# EPICS autosave request: apps/xpsMotorApp/Db/hpsSvtTopScan.req
$(PREF)hps:svt_top:motor:scan1.P1PA
$(PREF)hps:svt_top:motor:scan1.P1SM
$(PREF)hps:svt_top:motor:scan1.P1SP
$(PREF)hps:svt_top:motor:scan1.P1EP
$(PREF)hps:svt_top:motor:scan1.NPTS
$(PREF)hps:svt_top:motor:saveData_scanNumber
$(PREF)hps:svt_top:motor:saveData_fileSystem
$(PREF)hps:svt_top:motor:saveData_subDir
$(PREF)hps:svt_top:motor:saveData_baseName
$(PREF)hps:svt_top:motor:scan1.PDLY
$(PREF)hps:svt_top:motor:scan1.DDLY
$(PREF)hps:svt_top:motor:scan1.PASM
